INTERFACE I_State

METHOD Execute
END_METHOD

PROPERTY Name : STRING
GET
END_GET
END_PROPERTY

METHOD OnEntry
END_METHOD

METHOD OnExit
END_METHOD

END_INTERFACE

(* stored: Version 1.1.0.1, ProductVersion 3.1.4024.12
   Itf I_State: Id {ffd42d10-eba7-0ded-0838-25f0e9b01e95}
   Method Execute: Id {339f8b31-fc52-004c-17f6-c628a14c29f9}
   Property Name: Id {89adc5fb-2e73-0650-306e-70919788ddc6}
   Get Get: Id {65df2e94-70c8-04c9-03fc-4a256b782655}
   Method OnEntry: Id {0cb9de10-47c6-0557-2a8b-0d981bd44305}
   Method OnExit: Id {147f60a6-0f6f-0957-0b01-dc21ca030f56} *)
